TYPE ST_XTS_TRANSPORT_CTRL :
STRUCT
  Cmd       : E_XTS_TRANSPORT_CTRL;
END_STRUCT
END_TYPE

(* stored: Version 1.1.0.1, ProductVersion 3.1.4024.12
   DUT ST_XTS_TRANSPORT_CTRL: Id {4a457e1d-235c-4b07-b217-e2343bd64c6b} *)
